INTERFACE I_ExternalLogger

METHOD AddToLog
VAR_IN_OUT
   Message : T_MaxString;
END_VAR
VAR_INPUT
   LogSeverity : E_LogSeverity;
END_VAR
END_METHOD

END_INTERFACE

(* stored: Version 1.1.0.1, ProductVersion 3.1.4024.9
   Itf I_ExternalLogger: Id {c359840c-cfe2-45ce-9a5a-254a11158f8f}
   Method AddToLog: Id {61706da7-0ed7-45c8-b0e5-d47f4fea8c64} *)
